(* CoDeSys 2.3.9.31 project: myhome.pro *)
(* Libraries: TcSUPS.lib 22.3.10 14:59:22, TcBaseMath.lib 27.7.04 13:07:56, TcMath.lib 23.9.04 16:15:30, TcBABasic.lib 29.5.12 16:01:34, TcBase.lib 14.5.09 13:14:08, TcSystem.lib 27.2.12 16:08:36, TcUtilities.lib 2.3.12 20:25:40, TcEL6851.lib 22.4.12 13:04:27, STANDARD.LIB 5.6.98 13:03:02, TcpIp.lib 13.10.11 11:31:34, beckhoff_network_121.lib 6.5.14 22:11:45, oscat_basic_333.lib 6.5.14 22:41:24 *)

(* Global variable list: Global_Variables *)
VAR_GLOBAL

	SYS_VKE_0:		BOOL	:=	FALSE;		(*SYSTEM ALWAYS 0*)
	SYS_VKE_1:		BOOL	:=	TRUE;		(*SYSTEM ALWAYS 1*)
	SYS_IBN_1:		BOOL	:=	TRUE;		(*SYSTEM IBN ALWAYS 1*)

	di_System_Time:	DINT;

	SYS_FPE_100MS:	BOOL	:=	FALSE;		(*SYSTEM TIME 0.1 sec*)
	SYS_FPE_200MS:	BOOL	:=	FALSE;		(*SYSTEM TIME 0.2 sec*)
	SYS_FPE_500MS:	BOOL	:=	FALSE;		(*SYSTEM TIME 0.5 sec*)
	SYS_FPE_1S:		BOOL	:=	FALSE;		(*SYSTEM TIME 1.0 sec*)
	SYS_FPE_2S:		BOOL	:=	FALSE;		(*SYSTEM TIME 2.0 sec*)

	SYS_TOG_100MS:	BOOL	:=	FALSE;		(*SYSTEM TIME 0.1 sec*)
	SYS_TOG_200MS:	BOOL	:=	FALSE;		(*SYSTEM TIME 0.2 sec*)
	SYS_TOG_500MS:	BOOL	:=	FALSE;		(*SYSTEM TIME 0.5 sec*)
	SYS_TOG_1S:		BOOL	:=	FALSE;		(*SYSTEM TIME 1.0 sec*)
	SYS_TOG_2S:		BOOL	:=	FALSE;		(*SYSTEM TIME 2.0 sec*)

	SYS_T_100MS:		TON;					(*SYSTEM TIME 0.1 sec*)
	SYS_T_200MS:		TON;					(*SYSTEM TIME 0.2 sec*)
	SYS_T_500MS:		TON;					(*SYSTEM TIME 0.5 sec*)
	SYS_T_1S:			TON;					(*SYSTEM TIME 1.0 sec*)
	SYS_T_2S:			TON;					(*SYSTEM TIME 2.0 sec*)

	AX_FPE_100MS:	R_TRIG;				(*SYSTEM AUX FPE 0.1 sec*)
	AX_FPE_200MS:	R_TRIG;				(*SYSTEM AUX FPE 0.2 sec*)
	AX_FPE_500MS:	R_TRIG;				(*SYSTEM AUX FPE 0.5 sec*)
	AX_FPE_1S:		R_TRIG;				(*SYSTEM AUX FPE 1.0 sec*)
	AX_FPE_2S:		R_TRIG;				(*SYSTEM AUX FPE 2.0 sec*)

(*DIGITAL INPUTS/Outputs*)
	(*SPS Switch 01 Arbeitsraum*)
	DI_S01_1 	AT %IX50.0 : BOOL;	(*Function Left 1*)
	DI_S01_2	AT %IX50.1 : BOOL;	(*Function Right 1*)
	DI_S01_3	AT %IX50.2 : BOOL;	(*Function Left 2*)
	DI_S01_4	AT %IX50.3 : BOOL;	(*Function Right 2*)
	DI_S01_5	AT %IX50.4 : BOOL;	(*Function Left 3*)
	DI_S01_6	AT %IX50.5 : BOOL;	(*Function Right 3*)
	DO_S01_0 	AT %QX50.0 : BOOL;	(*Status LED Left 1*)
	DO_S01_1 	AT %QX50.1 : BOOL;	(*Status LED Right 1*)
	DO_S01_2 	AT %QX50.2 : BOOL;	(*Status LED Left 2*)
	DO_S01_3 	AT %QX50.3 : BOOL;	(*Status LED Right 2*)
	DO_S01_4 	AT %QX50.4 : BOOL;	(*Status LED Left 3*)
	DO_S01_5 	AT %QX50.5 : BOOL;	(*Status LED Right 3*)
	DO_S01_6 	AT %QX50.6 : BOOL;	(*Background LED*)

	(*SPS Switch 02 Wohnzimmer*)
	DI_S02_1 	AT %IX50.6 : BOOL;	(*Function Left 1*)
	DI_S02_2	AT %IX50.7 : BOOL;	(*Function Right 1*)
	DI_S02_3	AT %IX51.0 : BOOL;	(*Function Left 2*)
	DI_S02_4	AT %IX51.1 : BOOL;	(*Function Right 2*)
	DI_S02_5	AT %IX51.2 : BOOL;	(*Function Left 3*)
	DI_S02_6	AT %IX51.3 : BOOL;	(*Function Right 3*)
	DO_S02_0 	AT %QX50.7 : BOOL;	(*Status LED Left 1*)
	DO_S02_1 	AT %QX51.0 : BOOL;	(*Status LED Right 1*)
	DO_S02_2 	AT %QX51.1 : BOOL;	(*Status LED Left 2*)
	DO_S02_3 	AT %QX51.2 : BOOL;	(*Status LED Right 2*)
	DO_S02_4 	AT %QX51.3 : BOOL;	(*Status LED Left 3*)
	DO_S02_5 	AT %QX51.4 : BOOL;	(*Status LED Right 3*)
	DO_S02_6 	AT %QX51.5 : BOOL;	(*Background LED*)

	(*DOUBLE Switch 03*)
	DI_S03_1 	AT %IX51.4 : BOOL;	(*Function Left*)
	DI_S03_2 	AT %IX51.5 : BOOL;	(*Function Right*)

	(*DOUBLE Switch 04*)
	DI_S04_1 	AT %IX51.6 : BOOL;	(*Function Left*)
	DI_S04_2 	AT %IX51.7 : BOOL;	(*Function Right*)

	(*SPS Switch 05 Schlafzimmer Bett Links*)
	DI_S05_1 	AT %IX52.0 : BOOL;	(*Function Left 1*)
	DI_S05_2	AT %IX52.1 : BOOL;	(*Function Right 1*)
	DI_S05_3	AT %IX52.2 : BOOL;	(*Function Left 2*)
	DI_S05_4	AT %IX52.3 : BOOL;	(*Function Right 2*)
	DI_S05_5	AT %IX52.4 : BOOL;	(*Function Left 3*)
	DI_S05_6	AT %IX52.5 : BOOL;	(*Function Right 3*)
	DO_S05_0 	AT %QX51.6 : BOOL;	(*Status LED Left 1*)
	DO_S05_1 	AT %QX51.7 : BOOL;	(*Status LED Right 1*)
	DO_S05_2 	AT %QX52.0 : BOOL;	(*Status LED Left 2*)
	DO_S05_3 	AT %QX52.1 : BOOL;	(*Status LED Right 2*)
	DO_S05_4 	AT %QX52.2 : BOOL;	(*Status LED Left 3*)
	DO_S05_5 	AT %QX52.3 : BOOL;	(*Status LED Right 3*)
	DO_S05_6 	AT %QX52.4 : BOOL;	(*Background LED*)

	(*SPS Switch 06 Schlafzimmer Bett Rechts*)
	DI_S06_1 	AT %IX52.6 : BOOL;	(*Function Left 1*)
	DI_S06_2	AT %IX52.7 : BOOL;	(*Function Right 1*)
	DI_S06_3	AT %IX53.0 : BOOL;	(*Function Left 2*)
	DI_S06_4	AT %IX53.1 : BOOL;	(*Function Right 2*)
	DI_S06_5	AT %IX53.2 : BOOL;	(*Function Left 3*)
	DI_S06_6	AT %IX53.3 : BOOL;	(*Function Right 3*)
	DO_S06_0 	AT %QX52.5 : BOOL;	(*Status LED Left 1*)
	DO_S06_1 	AT %QX52.6 : BOOL;	(*Status LED Right 1*)
	DO_S06_2 	AT %QX52.7 : BOOL;	(*Status LED Left 2*)
	DO_S06_3 	AT %QX53.0 : BOOL;	(*Status LED Right 2*)
	DO_S06_4 	AT %QX53.1 : BOOL;	(*Status LED Left 3*)
	DO_S06_5 	AT %QX53.2 : BOOL;	(*Status LED Right 3*)
	DO_S06_6 	AT %QX53.3 : BOOL;	(*Background LED*)

	(*DOUBLE Switch 07*)
	DI_S07_1 	AT %IX53.4 : BOOL;	(*Function Left*)
	DI_S07_2 	AT %IX53.5 : BOOL;	(*Function Right*)

	(*SINGLE Switch 08*)
	DI_S08	 	AT %IX53.6 : BOOL;	(*Function*)

	(*SINGLE Switch 09*)
	DI_S09	 	AT %IX53.7 : BOOL;	(*Function*)

	(*SINGLE Switch 10*)
	DI_S10	 	AT %IX54.0 : BOOL;	(*Function*)

	(*SINGLE Swith 11*)
	DI_S11	 	AT %IX54.1 : BOOL;	(*Function*)

	(*Relais*)
	DO_NN_K01	AT %QX54.0 : BOOL;	(*Relais Netzteil Arbeitsraum*)
	DO_NN_K02	AT %QX54.1 : BOOL;	(*Relais Steckdosen Arbeitsraum*)
	DO_NN_K03	AT %QX54.2 : BOOL;	(*Relais Netzteil Wohnzimmer*)
	DO_NN_K04	AT %QX54.3 : BOOL;	(*Relais Steckdosen Fernseher*)
	DO_NN_K05	AT %QX54.4 : BOOL;	(*Relais Netzteil Küche*)
	DO_NN_K06	AT %QX54.5 : BOOL;	(*Relais Netzteil Zimmer / Schlafzimmer*)
	DO_NN_K07	AT %QX54.6 : BOOL;	(*Relais Netzteil WC, Gang und Abstellraum*)
	DO_NN_K08	AT %QX54.7 : BOOL;	(*Relais Reserve*)
	DO_NN_K09	AT %QX53.6 : BOOL;	(*Relais Reserve*)
	DO_NN_K10	AT %QX53.7 : BOOL;	(*Relais Reserve*)

(* DMX Line *)
	fbEL6851Communication	:	FB_EL6851Communication;
	stDMXInDataLinie01               AT %I*	:	ST_EL6851InData;
	stDMXOutDataLinie01              AT %Q*	:	ST_EL6851OutData;
	stCommandBuffer01						:	ST_DMXCommandBuffer;
	arrDMXProcessData						:	ARRAY [1..512] OF BYTE;

END_VAR

(* Global variable list: TwinCAT_Configuration *)
(* Generated automatically by TwinCAT - (read only) *)
VAR_CONFIG
	.stDMXInDataLinie01 AT %IB56 : ST_EL6851InData;
	.stDMXOutDataLinie01 AT %QB56 : ST_EL6851OutData;
END_VAR

(* Data type *)
TYPE Type_HSV :
STRUCT
	Hue	:			REAL;
	Saturation:		REAL:= 100.0;
	Brightness:		REAL:=100.0;
END_STRUCT
END_TYPE

(* Data type *)
TYPE Type_LED :
STRUCT
	Switch_ON:			BOOL;
	Switch_RANDOM:		BOOL;
	bLight:				BOOL;
	Config:				Type_LED_CONFIG;
	Value:				REAL:=100;
	Brightness:			BYTE;
	fbDimmer2Switch: FB_Dimmer2Switch;
	fpSwitchOnOff: F_TRIG;
END_STRUCT
END_TYPE

(* Data type *)
TYPE Type_LED_CONFIG :
STRUCT
	tDimmTime: 		REAL	:= 5000;
	bDimmOnMode:	BOOL	:= TRUE;
	tDimmOnTime:		REAL	:= 500;
	bDimmOffMode:	BOOL	:= TRUE;
	tDimmOffTime:		REAL	:= 1000;
	Brightness_MAX	:REAL:=255;
END_STRUCT
END_TYPE

(* Data type *)
TYPE Type_LED_RGB :
STRUCT
	Hue				:REAL;
	Saturation			:REAL:= 100.0;
	Brightness			:REAL:=100;
	Switch_ON			:BOOL;
	Switch_RANDOM	:BOOL;
	bLight:			BOOL;
	Config				:Type_LED_RGB_CONFIG;
	Red					:BYTE;
	Green				:BYTE;
	Blue					:BYTE;
	fbDimmer2Switch: FB_Dimmer2Switch;
	fpSwitchOnOff: F_TRIG;
END_STRUCT
END_TYPE

(* Data type *)
TYPE Type_LED_RGB_CONFIG :
STRUCT
	Speed_RANDOM	:REAL;

	tDimmTime: 		REAL	:= 5000;
	bDimmOnMode:	BOOL	:= TRUE;
	tDimmOnTime:		REAL	:= 500;
	bDimmOffMode:	BOOL	:= TRUE;
	tDimmOffTime:		REAL	:= 1000;
END_STRUCT
END_TYPE

(* Data type *)
TYPE Type_SCENE_CONFIG :
STRUCT
	tDimmTime: 		REAL	:= 5000;
	bDimmOnMode:	BOOL	:= TRUE;
	tDimmOnTime:		REAL	:= 500;
	bDimmOffMode:	BOOL	:= TRUE;
	tDimmOffTime:		REAL	:= 1000;
END_STRUCT
END_TYPE

(* Data type *)
TYPE Type_SCENE_WZ :
STRUCT
	bSceneActive:			BOOL;
	byWhiteUpNorth:			BYTE;
	byWhiteUpWest:			BYTE;
	byWhiteUpSouthEast:		BYTE;
	byWhiteMiddleNorthWest:	BYTE;
	byWhiteMiddleSouthEast:	BYTE;
	byWhiteDownNorthWest:	BYTE;
	byWhiteDownSouthEast:	BYTE;
	tyHSVUp:				Type_HSV;
	tyHSVMiddle: 			Type_HSV;
	tyHSVDown: 				Type_HSV;
	tyConfig:					Type_SCENE_CONFIG;
END_STRUCT
END_TYPE

(* POU MAIN, ST *)
PROGRAM MAIN
VAR
	YahooWeatherAltlengbach: FB_WEATHER;
END_VAR
FC_00_BASICS();

(*Aufruf Wohnräume*)
FC_01_ARBEITSZIMMER();
FC_02_WOHNZIMMER();
FC_03_KUECHE();
FC_04_ZIMMER();
FC_05_WC_GANG();

(*YahooWeatherAltlengbach();*)

(*WORLD_WEATHER_test();*)
YAHOO_WEATHER_test();

fbEL6851Communication(	wSourceManufacturerID := 16#42_41,
						dwSourceDeviceID := 16#12_13_14_15,
						bEnableSendingData := TRUE,
						bSetCycleMode := TRUE,
						bSendDefaultData := FALSE,
						uiDataLength := 512,
						dwOptions := 0,
						stEL6851InData := stDMXInDataLinie01,
						stEL6851OutData := stDMXOutDataLinie01,
						stCommandBuffer := stCommandBuffer01,
						arrProcessData := arrDMXProcessData);
END_PROGRAM

(* POU Weather/FB_WEATHER, ST *)
FUNCTION_BLOCK FB_WEATHER
VAR_INPUT
END_VAR
VAR_OUTPUT
END_VAR
VAR
	FB_Weather_PLZ_3033: YAHOO_WEATHER;
	vBOOL: BOOL := FALSE;
	vIP_C : IP_C;
	vS_BUF : NETWORK_BUFFER;
	vR_BUF : NETWORK_BUFFER;
	vYW : YAHOO_WEATHER_DATA;
	vBUSY : BOOL;
	vDONE : BOOL;
	vERROR_C : DWORD;
	vERROR_T : BYTE;
END_VAR
FB_Weather_PLZ_3033(
	ACTIVATE:= vBOOL,
	UNITS:= FALSE,
	LOCATION:= '541490',
	IP_C:=vIP_C ,
	S_BUF:=vS_BUF ,
	R_BUF:=vR_BUF ,
	YW:= vYW,
	BUSY=> vBUSY,
	DONE=>vDONE ,
	ERROR_C=>vERROR_C ,
	ERROR_T=>vERROR_T );
END_FUNCTION_BLOCK

(* POU FC_00_BASICS, ST *)
PROGRAM FC_00_BASICS
VAR
	T_100ms_TON: TON;
	T_100ms_TOF: TOF;

(* UPS related ... *)
	fbUPS			: FB_S_UPS;			(* UPS-FB instance *)
					(* Default Values of FB_S_UPS-Inputs:
						sNetID 			:= '' ==> local netid
						iPLCPort 		:= AMSPORT_R0_PLC_RTS1 ==> 801 = 1st Runtime System
						iUPSPort		:= 16#4A8 ==> Port for reading Power State of UPS
						tTimeout 		:= DEFAULT_ADS_TIMEOUT ==> 5S
						eUpsMode 		:= eSUPS_WrPersistData_Shutdown ==> writing persistent data + shutdown
						ePersistentMode := SPDM_2PASS ==> All data is from same plc cycle, cycletime exceeds possible. Plc stops with the shutdown, a few cycles after writing persistent data. 
						tRecoverTime 	:= T#10s ==> 10s power to recover from short power failure before eSUPS_PowerOK is reported (in mode eSUPS_WrPersistData_NoShutdown/eSUPS_CheckPowerStatus)
					*)
	eUpsMode		: E_S_UPS_Mode	:= eSUPS_WrPersistData_Shutdown; (* UPS mode (writing persistent data + shutdown) *)

	(* !!! TO DO: REPLACE WITH YOUR PLC VARIABLES/FB INSTANCES !!! regular PLC variables/FB instances ... *)
	iCounter		: UDINT;					(* non persistent counter *)

END_VAR

VAR PERSISTENT
	(* !!! TO DO: REPLACE WITH YOUR PERSISTENT PLC VARIABLES !!! persistent variables ... *)
	iPowerFailureCount: UDINT:=0; (* persistent counter of power failures *)
END_VAR
SYS_VKE_0		:=	FALSE;
SYS_VKE_1		:=	TRUE;
SYS_IBN_1		:=	TRUE;

di_System_Time := TIME_TO_DINT(TIME());


(*GENERATE SYSTEM PULSE FLAGS*)

SYS_T_100MS(IN:= SYS_IBN_1 AND NOT SYS_T_100MS.Q, PT:= T#100MS);
SYS_T_200MS(IN:= SYS_IBN_1 AND NOT SYS_T_200MS.Q, PT:= T#200MS);
SYS_T_500MS(IN:= SYS_IBN_1 AND NOT SYS_T_500MS.Q, PT:= T#500MS);
SYS_T_1S(IN:= SYS_IBN_1 AND NOT SYS_T_1S.Q, PT:= T#1S);
SYS_T_2S(IN:= SYS_IBN_1 AND NOT SYS_T_2S.Q, PT:= T#2S);

IF SYS_T_100MS.Q	THEN
	IF SYS_TOG_100MS THEN
		SYS_TOG_100MS := FALSE; 	ELSE	SYS_TOG_100MS := TRUE;
	END_IF
END_IF

IF SYS_T_200MS.Q	THEN
	IF SYS_TOG_200MS THEN
		SYS_TOG_200MS := FALSE; 	ELSE	SYS_TOG_200MS := TRUE;
	END_IF
END_IF

IF SYS_T_500MS.Q	THEN
	IF SYS_TOG_500MS THEN
		SYS_TOG_500MS := FALSE; 	ELSE	SYS_TOG_500MS := TRUE;
	END_IF
END_IF

IF SYS_T_1S.Q	THEN
	IF SYS_TOG_1S THEN
		SYS_TOG_1S := FALSE; 	ELSE	SYS_TOG_1S := TRUE;
	END_IF
END_IF

IF SYS_T_2S.Q	THEN
	IF SYS_TOG_2S THEN
		SYS_TOG_2S := FALSE; 	ELSE	SYS_TOG_2S := TRUE;
	END_IF
END_IF

AX_FPE_100MS(CLK:= SYS_TOG_100MS , Q=> SYS_FPE_100MS);
AX_FPE_200MS(CLK:= SYS_TOG_200MS , Q=> SYS_FPE_200MS);
AX_FPE_500MS(CLK:= SYS_TOG_500MS , Q=> SYS_FPE_500MS);
AX_FPE_1S(CLK:= SYS_TOG_1S , Q=> SYS_FPE_1S);
AX_FPE_2S(CLK:= SYS_TOG_2S , Q=> SYS_FPE_2S);

(* S-UPS Demo *)

(* call UPS-FB instance in first lines of the fastest PLC Task *)
fbUPS(eUpsMode := eUpsMode);
(* eUpsMode =							in case of powerfailure:
	 eSUPS_WrPersistData_Shutdown 		 	writing of persistent data + shutdown
	 eSUPS_WrPersistData_NoShutdown 		writing of PERSISTENT data, no shutdown
	 eSUPS_CheckPowerStatus 				reports powerfailure without ACTION (no writing, no shutdown) 
	 eSUPS_ImmediateShutdown 				skips writing of data, immediate shutdown
*)

(* evaluate UPS State *)
IF eGlobalSUpsState = eSUPS_PowerFailure THEN
	(* first cycle of powerfailure *)

	(* execute code that should only be done once with each powerfailure, i.e. increase powerfailure counter *)
	iPowerFailureCount := iPowerFailureCount + 1;
END_IF
END_PROGRAM

(* POU FC_01_ARBEITSZIMMER, ST *)
PROGRAM FC_01_ARBEITSZIMMER
VAR PERSISTENT
	tyWhiteCeiling:			Type_LED;
	tyWhiteWorkplace:		Type_LED;
	tyWhiteRegal:			Type_LED;
	tyWhiteAbstellraum:		Type_LED;
	tyWhiteReserve1:			Type_LED;
	tyWhiteReserve2:			Type_LED;
	tyWhiteReserve3:			Type_LED;
	tyWhiteReserve4:			Type_LED;
END_VAR
(*LED light white ceiling*)
PRG_LED_SINGLECOLOR(
	i_bSwitchOn:= DI_S01_1,
	i_bSwitchOff:= FALSE,
	i_bSwitchOnOff:= DI_S01_1,
	i_iSceneValue:= ,
	io_TypeLED:= tyWhiteCeiling);

(*LED light white workplace*)
PRG_LED_SINGLECOLOR(
	i_bSwitchOn:= DI_S01_1,
	i_bSwitchOff:= FALSE,
	i_bSwitchOnOff:= FALSE,
	i_iSceneValue:= ,
	io_TypeLED:= tyWhiteWorkplace);

(*LED light white Regal*)
PRG_LED_SINGLECOLOR(
	i_bSwitchOn:= FALSE,
	i_bSwitchOff:= FALSE,
	i_bSwitchOnOff:= FALSE,
	i_iSceneValue:= ,
	io_TypeLED:= tyWhiteRegal);

(*LED light white Abstellraum*)
PRG_LED_SINGLECOLOR(
	i_bSwitchOn:= FALSE,
	i_bSwitchOff:= FALSE,
	i_bSwitchOnOff:= FALSE,
	i_iSceneValue:= ,
	io_TypeLED:= tyWhiteAbstellraum);

(*LED light white Reserve*)
PRG_LED_SINGLECOLOR(
	i_bSwitchOn:= FALSE,
	i_bSwitchOff:= FALSE,
	i_bSwitchOnOff:= FALSE,
	i_iSceneValue:= ,
	io_TypeLED:= tyWhiteReserve1);

(*LED light white Reserve*)
PRG_LED_SINGLECOLOR(
	i_bSwitchOn:= FALSE,
	i_bSwitchOff:= FALSE,
	i_bSwitchOnOff:= FALSE,
	i_iSceneValue:= ,
	io_TypeLED:= tyWhiteReserve2);

(*LED light white Reserve*)
PRG_LED_SINGLECOLOR(
	i_bSwitchOn:= FALSE,
	i_bSwitchOff:= FALSE,
	i_bSwitchOnOff:= FALSE,
	i_iSceneValue:= ,
	io_TypeLED:= tyWhiteReserve3);

(*LED light white Reserve*)
PRG_LED_SINGLECOLOR(
	i_bSwitchOn:= FALSE,
	i_bSwitchOff:= FALSE,
	i_bSwitchOnOff:= FALSE,
	i_iSceneValue:= ,
	io_TypeLED:= tyWhiteReserve4);

(*relay for power supply*)
DO_NN_K01 :=	tyWhiteCeiling.bLight OR tyWhiteWorkplace.bLight OR tyWhiteRegal.bLight OR
				tyWhiteAbstellraum.bLight OR tyWhiteReserve1.bLight OR tyWhiteReserve2.bLight OR
				tyWhiteReserve3.bLight OR tyWhiteReserve4.bLight;
(*DMX communication*)
arrDMXProcessData[1] := tyWhiteCeiling.Brightness;
arrDMXProcessData[2] := tyWhiteWorkplace.Brightness;
arrDMXProcessData[3] := tyWhiteRegal.Brightness;
arrDMXProcessData[4] := tyWhiteAbstellraum.Brightness;
arrDMXProcessData[5] := tyWhiteReserve1.Brightness;
arrDMXProcessData[6] := tyWhiteReserve2.Brightness;
arrDMXProcessData[7] := tyWhiteReserve3.Brightness;
arrDMXProcessData[8] := tyWhiteReserve4.Brightness;
END_PROGRAM

(* POU PRG_LED_SINGLECOLOR, ST *)
PROGRAM PRG_LED_SINGLECOLOR
VAR_INPUT
	i_bSwitchOn:		BOOL;
	i_bSwitchOff:		BOOL;
	i_bSwitchOnOff:	BOOL;
	i_iSceneValue:	INT;
END_VAR

VAR_IN_OUT
	io_TypeLED: Type_LED;		(*CONTAINS THE LIGHT STATUS*)
END_VAR
(*flag positive edge of switch for on and off*)
io_TypeLED.fpSwitchOnOff(CLK:= i_bSwitchOnOff );

(*switch light on*)
IF i_bSwitchOn OR (io_TypeLED.fpSwitchOnOff.Q AND NOT io_TypeLED.bLight) THEN
	io_TypeLED.Switch_ON := TRUE;
END_IF

(*switch light off*)
IF i_bSwitchOff OR (io_TypeLED.fpSwitchOnOff.Q AND io_TypeLED.bLight) THEN
	io_TypeLED.Switch_ON := FALSE;
END_IF

io_TypeLED.fbDimmer2Switch(
	bSwitchDimmUp:= FALSE,
	bSwitchDimmDown:= FALSE,
	bOn:= io_TypeLED.Switch_ON,
	bOff:= NOT io_TypeLED.Switch_ON,
	bSetDimmValue:= FALSE,
	nDimmValue:= 0,
	tSwitchOverTime:=T#300MS ,
	tDimmTime:= REAL_TO_TIME(io_TypeLED.Config.tDimmTime),
	bMemoryModeOn:= TRUE,
	nOnValueWithoutMemoryMode:= 0,
	bDimmOnMode:= io_TypeLED.Config.bDimmOnMode,
	tDimmOnTime:= REAL_TO_TIME(io_TypeLED.Config.tDimmOnTime),
	bDimmOffMode:= io_TypeLED.Config.bDimmOffMode,
	tDimmOffTime:= REAL_TO_TIME(io_TypeLED.Config.tDimmOffTime),
	nOutMin:= 0,
	nOutMax:=100,
	bLight=> io_TypeLED.bLight);

io_TypeLED.Brightness := REAL_TO_BYTE(UINT_TO_REAL(io_TypeLED.fbDimmer2Switch.nOut)/100*io_TypeLED.Config.Brightness_MAX*(io_TypeLED.Value/100));
END_PROGRAM

(* POU FC_02_WOHNZIMMER, ST *)
PROGRAM FC_02_WOHNZIMMER
VAR PERSISTENT
	tyScene1: Type_SCENE_WZ;
	tyScene2: Type_SCENE_WZ;
	tyScene3: Type_SCENE_WZ;
	tyScene4: Type_SCENE_WZ;
	tyScene5: Type_SCENE_WZ;
	tyScene6: Type_SCENE_WZ;
	tyScene7: Type_SCENE_WZ;
	tyScene8: Type_SCENE_WZ;
	tyScene9: Type_SCENE_WZ;
	tyScene10: Type_SCENE_WZ;
	tyScene11: Type_SCENE_WZ;
	tyScene12: Type_SCENE_WZ;
	tyScene13: Type_SCENE_WZ;
	tyScene14: Type_SCENE_WZ;
	tyScene15: Type_SCENE_WZ;

	tyActScene:Type_SCENE_WZ;

	tyWhiteUpNorth:				Type_LED;
	tyWhiteUpWest:				Type_LED;
	tyWhiteUpSouthEast:			Type_LED;
	tyWhiteMiddleNorthWest:		Type_LED;
	tyWhiteMiddleSouthEast:		Type_LED;
	tyWhiteDownNorthWest:		Type_LED;
	tyWhiteDownSouthEast:		Type_LED;
	tyRGBUp:					Type_LED_RGB;
	tyRGBMiddle: 				Type_LED_RGB;
	tyRGBDown: 					Type_LED_RGB;

END_VAR
(*Scene control*)
PRG_SCENE_CONTROL_WZ(
	i_bNextScene:= , 
	i_bPrevScene:= , 
	io_tyScene1:= tyScene1,
	io_tyScene2:= tyScene2,
	io_tyScene3:= tyScene3,
	io_tyScene4:= tyScene4,
	io_tyScene5:= tyScene5,
	io_tyScene6:= tyScene6,
	io_tyScene7:= tyScene7,
	io_tyScene8:= tyScene8,
	io_tyScene9:= tyScene9,
	io_tyScene10:= tyScene10,
	io_tyScene11:= tyScene11,
	io_tyScene12:= tyScene12,
	io_tyScene13:= tyScene13,
	io_tyScene14:= tyScene14,
	io_tyScene15:= tyScene15,
	o_tyActScene=> tyActScene);

(*LED light white up north*)
PRG_LED_SINGLECOLOR(
	i_bSwitchOn:= FALSE,
	i_bSwitchOff:= FALSE,
	i_bSwitchOnOff:= FALSE,
	i_iSceneValue:= tyActScene.byWhiteUpNorth,
	io_TypeLED:= tyWhiteUpNorth);

(*LED light white up west*)
PRG_LED_SINGLECOLOR(
	i_bSwitchOn:= FALSE,
	i_bSwitchOff:= FALSE,
	i_bSwitchOnOff:= FALSE,
	i_iSceneValue:= tyActScene.byWhiteUpWest,
	io_TypeLED:= tyWhiteUpWest);

(*LED light white up southeast*)
PRG_LED_SINGLECOLOR(
	i_bSwitchOn:= FALSE,
	i_bSwitchOff:= FALSE,
	i_bSwitchOnOff:=FALSE ,
	i_iSceneValue:= tyActScene.byWhiteUpSouthEast,
	io_TypeLED:= tyWhiteUpSouthEast);

(*LED light white middle northwest*)
PRG_LED_SINGLECOLOR(
	i_bSwitchOn:= FALSE,
	i_bSwitchOff:= FALSE,
	i_bSwitchOnOff:= FALSE,
	i_iSceneValue:= tyActScene.byWhiteMiddleNorthWest,
	io_TypeLED:= tyWhiteMiddleNorthWest);

(*LED light white middle southeast*)
PRG_LED_SINGLECOLOR(
	i_bSwitchOn:= FALSE,
	i_bSwitchOff:= FALSE,
	i_bSwitchOnOff:= FALSE,
	i_iSceneValue:= tyActScene.byWhiteMiddleSouthEast,
	io_TypeLED:= tyWhiteMiddleSouthEast);

(*LED light white down northwest*)
PRG_LED_SINGLECOLOR(
	i_bSwitchOn:= FALSE,
	i_bSwitchOff:= FALSE,
	i_bSwitchOnOff:=FALSE ,
	i_iSceneValue:= tyActScene.byWhiteDownNorthWest,
	io_TypeLED:= tyWhiteDownNorthWest);

(*LED light white down southeast*)
PRG_LED_SINGLECOLOR(
	i_bSwitchOn:= FALSE,
	i_bSwitchOff:= FALSE,
	i_bSwitchOnOff:= FALSE,
	i_iSceneValue:= tyActScene.byWhiteDownSouthEast,
	io_TypeLED:= tyWhiteDownSouthEast);

(*LED light RGB upper row*)
PRG_LED_MULTICOLOR(
	i_SwitchON:= FALSE,
	i_SwitchOFF:= FALSE,
	i_bSwitchOnOff:= DI_S02_3,
	i_iSceneValue:= ,
	di_SysTime:= di_System_Time,
	io_Type_LED_RGB:= tyRGBUp);

(*LED light RGB middle row*)
PRG_LED_MULTICOLOR(
	i_SwitchON:= FALSE,
	i_SwitchOFF:= FALSE,
	i_bSwitchOnOff:= FALSE,
	i_iSceneValue:= ,
	di_SysTime:= di_System_Time,
	io_Type_LED_RGB:= tyRGBMiddle);

(*LED light RGB bottom row*)
PRG_LED_MULTICOLOR(
	i_SwitchON:= FALSE,
	i_SwitchOFF:= FALSE,
	i_bSwitchOnOff:= FALSE,
	i_iSceneValue:= ,
	di_SysTime:=di_System_Time ,
	io_Type_LED_RGB:= tyRGBDown);

(*relay for power supply*)
DO_NN_K03:=	tyWhiteUpNorth.bLight OR tyWhiteUpWest.bLight OR tyWhiteUpSouthEast.bLight OR
				tyWhiteMiddleNorthWest.bLight OR tyWhiteMiddleSouthEast.bLight OR tyWhiteDownNorthWest.bLight OR
				tyWhiteDownSouthEast.bLight OR tyRGBUp.bLight OR tyRGBMiddle.bLight OR tyRGBDown.bLight;

(*DMX communication*)
arrDMXProcessData[10] := tyWhiteUpNorth.Brightness;
arrDMXProcessData[11] := tyWhiteUpWest.Brightness;
arrDMXProcessData[12] := tyWhiteUpSouthEast.Brightness;
arrDMXProcessData[13] := tyWhiteMiddleNorthWest.Brightness;
arrDMXProcessData[14] := tyWhiteMiddleSouthEast.Brightness;
arrDMXProcessData[15] := tyWhiteDownNorthWest.Brightness;
arrDMXProcessData[16] := tyWhiteDownSouthEast.Brightness;
arrDMXProcessData[17] := tyRGBUp.Red;
arrDMXProcessData[18] := tyRGBUp.Green;
arrDMXProcessData[19] := tyRGBUp.Blue;
arrDMXProcessData[20] := tyRGBMiddle.Red;
arrDMXProcessData[21] := tyRGBMiddle.Green;
arrDMXProcessData[22] := tyRGBMiddle.Blue;
arrDMXProcessData[23] := tyRGBDown.Red;
arrDMXProcessData[24] := tyRGBDown.Green;
arrDMXProcessData[25] := tyRGBDown.Blue;
END_PROGRAM

(* POU PRG_SCENE_CONTROL_WZ, ST *)
PROGRAM PRG_SCENE_CONTROL_WZ
VAR_INPUT
	i_bNextScene:	BOOL;
	i_bPrevScene:	BOOL;
END_VAR

VAR_IN_OUT
	io_tyScene1: Type_SCENE_WZ;
	io_tyScene2: Type_SCENE_WZ;
	io_tyScene3: Type_SCENE_WZ;
	io_tyScene4: Type_SCENE_WZ;
	io_tyScene5: Type_SCENE_WZ;
	io_tyScene6: Type_SCENE_WZ;
	io_tyScene7: Type_SCENE_WZ;
	io_tyScene8: Type_SCENE_WZ;
	io_tyScene9: Type_SCENE_WZ;
	io_tyScene10: Type_SCENE_WZ;
	io_tyScene11: Type_SCENE_WZ;
	io_tyScene12: Type_SCENE_WZ;
	io_tyScene13: Type_SCENE_WZ;
	io_tyScene14: Type_SCENE_WZ;
	io_tyScene15: Type_SCENE_WZ;
END_VAR

VAR_OUTPUT
	o_tyActScene: Type_SCENE_WZ;
END_VAR

VAR
	fpNextScene: F_TRIG;
	fpPrevScene: F_TRIG;
	v_iActScene:	INT	:= 1;
END_VAR
fpNextScene(CLK:=i_bNextScene);
fpPrevScene(CLK:=i_bPrevScene);

IF fpNextScene.Q THEN
	v_iActScene := v_iActScene + 1;
END_IF

IF fpPrevScene.Q THEN
	v_iActScene := v_iActScene - 1;
END_IF

IF v_iActScene >= 17 THEN
	v_iActScene := 1;
END_IF

IF v_iActScene <= 0 THEN
	v_iActScene := 16;
END_IF

o_tyActScene := io_tyScene1;

CASE v_iActScene OF
1:	o_tyActScene := io_tyScene1;
2:	o_tyActScene := io_tyScene2;
3:	o_tyActScene := io_tyScene3;
4:	o_tyActScene := io_tyScene4;
5:	o_tyActScene := io_tyScene5;
6:	o_tyActScene := io_tyScene6;
7:	o_tyActScene := io_tyScene7;
8:	o_tyActScene := io_tyScene8;
9:	o_tyActScene := io_tyScene9;
10:	o_tyActScene := io_tyScene10;
11:	o_tyActScene := io_tyScene11;
12:	o_tyActScene := io_tyScene12;
13:	o_tyActScene := io_tyScene13;
14:	o_tyActScene := io_tyScene14;
15:	o_tyActScene := io_tyScene15;
END_CASE
END_PROGRAM

(* POU PRG_LED_MULTICOLOR, ST *)
PROGRAM PRG_LED_MULTICOLOR
VAR_INPUT
	i_SwitchON:	BOOL;
	i_SwitchOFF:	BOOL;
	i_bSwitchOnOff:	BOOL;
	i_iSceneValue:	INT;
	di_SysTime:	DINT;
END_VAR

VAR
	v_HUE: REAL;
	v_SATURATION: REAL;
	v_VALUE: REAL;
	v_RED: BYTE;
	v_GREEN: BYTE;
	v_BLUE: BYTE;
	v_VAR_H: REAL;
	v_VAR_I: REAL;
	v_VAR_1: REAL;
	v_VAR_2: REAL;
	v_VAR_3: REAL;
	v_VAR_R: REAL;
	v_VAR_G: REAL;
	v_VAR_B: REAL;
	v_Sys_Time_last_Call:	DINT;
	v_Cycle_Time:	DINT;

END_VAR
VAR_IN_OUT
	io_Type_LED_RGB: Type_LED_RGB;		(*CONTAINS THE LIGHT STATUS*)
END_VAR
(*Calculate the System Time between the last and the actual cycle for automatic color switching*)
v_Cycle_Time := di_SysTime - v_Sys_Time_last_Call;
v_Sys_Time_last_Call := di_SysTime;

(*flag positive edge of switch for on and off*)
io_Type_LED_RGB.fpSwitchOnOff(CLK:= i_bSwitchOnOff );

(*switch light on*)
IF i_SwitchON OR (io_Type_LED_RGB.fpSwitchOnOff.Q AND NOT io_Type_LED_RGB.bLight) THEN
	io_Type_LED_RGB.Switch_ON := TRUE;
END_IF

(*switch light off*)
IF i_SwitchOFF OR (io_Type_LED_RGB.fpSwitchOnOff.Q AND io_Type_LED_RGB.bLight) THEN
	io_Type_LED_RGB.Switch_ON := FALSE;
END_IF

(*control light with standard FB from Beckhoff BaBasic Library*)
io_Type_LED_RGB.fbDimmer2Switch(
	bSwitchDimmUp:= FALSE,
	bSwitchDimmDown:= FALSE,
	bOn:= io_Type_LED_RGB.Switch_ON,
	bOff:= NOT io_Type_LED_RGB.Switch_ON,
	bSetDimmValue:= FALSE,
	nDimmValue:= 0,
	tSwitchOverTime:=T#300MS ,
	tDimmTime:= REAL_TO_TIME(io_Type_LED_RGB.Config.tDimmTime),
	bMemoryModeOn:= TRUE,
	nOnValueWithoutMemoryMode:= 0,
	bDimmOnMode:= io_Type_LED_RGB.Config.bDimmOnMode,
	tDimmOnTime:= REAL_TO_TIME(io_Type_LED_RGB.Config.tDimmOnTime),
	bDimmOffMode:= io_Type_LED_RGB.Config.bDimmOffMode,
	tDimmOffTime:= REAL_TO_TIME(io_Type_LED_RGB.Config.tDimmOffTime),
	nOutMin:= 0,
	nOutMax:=REAL_TO_UINT( io_Type_LED_RGB.Brightness),
	bLight=> io_Type_LED_RGB.bLight);

IF io_Type_LED_RGB.Config.Speed_RANDOM < 1000 THEN
	io_Type_LED_RGB.Config.Speed_RANDOM := 1000;
END_IF

IF io_Type_LED_RGB.Switch_RANDOM THEN
	io_Type_LED_RGB.Hue := io_Type_LED_RGB.Hue + 360/(io_Type_LED_RGB.Config.Speed_RANDOM)*DINT_TO_REAL(v_Cycle_Time);

	IF io_Type_LED_RGB.Hue >= 360 THEN
		io_Type_LED_RGB.Hue := io_Type_LED_RGB.Hue-360;
	END_IF
	IF io_Type_LED_RGB.Hue < 0 THEN
		io_Type_LED_RGB.Hue := 0;
	END_IF
END_IF

v_HUE := io_Type_LED_RGB.Hue / 360;
v_SATURATION := io_Type_LED_RGB.Saturation / 100;
v_VALUE := (io_Type_LED_RGB.Brightness*UINT_TO_REAL(io_Type_LED_RGB.fbDimmer2Switch.nOut)/100) / 100;

IF v_SATURATION = 0 THEN
	v_RED := REAL_TO_BYTE(v_VALUE * 255);
	v_GREEN := REAL_TO_BYTE(v_VALUE * 255);
	v_BLUE := REAL_TO_BYTE(v_VALUE * 255);
ELSE
	v_VAR_H := v_HUE * 6;
	v_VAR_I := FLOOR(REAL_TO_LREAL(v_VAR_H));
	v_VAR_1:= v_VALUE * (1 - v_SATURATION);
	v_VAR_2:= v_VALUE * (1 - v_SATURATION * (v_VAR_H - v_VAR_I));
	v_VAR_3:= v_VALUE * (1 - v_SATURATION * (1 - (v_VAR_H - v_VAR_I)));

	CASE REAL_TO_INT(v_VAR_I) OF
	0:
		v_VAR_R := v_VALUE;
		v_VAR_G := v_VAR_3;
		v_VAR_B := v_VAR_1;
	1:
		v_VAR_R := v_VAR_2;
		v_VAR_G := v_VALUE;
		v_VAR_B := v_VAR_1;
	2:
		v_VAR_R := v_VAR_1;
		v_VAR_G := v_VALUE;
		v_VAR_B := v_VAR_3;
	3:
		v_VAR_R := v_VAR_1;
		v_VAR_G := v_VAR_2;
		v_VAR_B := v_VALUE;
	4:
		v_VAR_R := v_VAR_3;
		v_VAR_G := v_VAR_1;
		v_VAR_B := v_VALUE;
	ELSE
		v_VAR_R := v_VALUE;
		v_VAR_G := v_VAR_1;
		v_VAR_B := v_VAR_2;
	END_CASE

	v_RED := REAL_TO_BYTE(v_VAR_R * 255);
	v_GREEN := REAL_TO_BYTE(v_VAR_G * 255);
	v_BLUE := REAL_TO_BYTE(v_VAR_B * 255);
END_IF

io_Type_LED_RGB.Red := v_RED;
io_Type_LED_RGB.Green := v_GREEN;
io_Type_LED_RGB.Blue := v_BLUE;
END_PROGRAM

(* POU FC_03_KUECHE, ST *)
PROGRAM FC_03_KUECHE
VAR PERSISTENT
	tyWhiteCeilingNorth:			Type_LED;
	tyWhiteCeilingSouth:			Type_LED;
	tyWhiteWorkplateNorth:		Type_LED;
	tyWhiteWorkplateSouth:		Type_LED;
	tyWhiteTableNorth:			Type_LED;
	tyWhiteTableSouth:			Type_LED;
END_VAR
(*LED light white ceiling north*)
PRG_LED_SINGLECOLOR(
	i_bSwitchOn:= FALSE,
	i_bSwitchOff:= FALSE,
	i_bSwitchOnOff:= FALSE,
	i_iSceneValue:= ,
	io_TypeLED:= tyWhiteCeilingNorth);

(*LED light white ceiling south*)
PRG_LED_SINGLECOLOR(
	i_bSwitchOn:= FALSE,
	i_bSwitchOff:= FALSE,
	i_bSwitchOnOff:= FALSE,
	i_iSceneValue:= ,
	io_TypeLED:= tyWhiteCeilingSouth);

(*LED light white workplate north*)
PRG_LED_SINGLECOLOR(
	i_bSwitchOn:= FALSE,
	i_bSwitchOff:= FALSE,
	i_bSwitchOnOff:= FALSE,
	i_iSceneValue:= ,
	io_TypeLED:= tyWhiteWorkplateNorth);

(*LED light white workplate south*)
PRG_LED_SINGLECOLOR(
	i_bSwitchOn:= FALSE,
	i_bSwitchOff:= FALSE,
	i_bSwitchOnOff:= FALSE,
	i_iSceneValue:= ,
	io_TypeLED:= tyWhiteWorkplateSouth);

(*LED light white table north*)
PRG_LED_SINGLECOLOR(
	i_bSwitchOn:= FALSE,
	i_bSwitchOff:= FALSE,
	i_bSwitchOnOff:= FALSE,
	i_iSceneValue:= ,
	io_TypeLED:= tyWhiteTableNorth);

(*LED light white table south*)
PRG_LED_SINGLECOLOR(
	i_bSwitchOn:= FALSE,
	i_bSwitchOff:= FALSE,
	i_bSwitchOnOff:= FALSE,
	i_iSceneValue:= ,
	io_TypeLED:= tyWhiteTableSouth);

(*relay for power supply*)
DO_NN_K05 :=	tyWhiteCeilingNorth.bLight OR tyWhiteCeilingSouth.bLight OR tyWhiteWorkplateNorth.bLight OR
				tyWhiteWorkplateSouth.bLight OR tyWhiteTableNorth.bLight OR tyWhiteTableSouth.bLight;

(*DMX communication*)
arrDMXProcessData[40] := tyWhiteCeilingNorth.Brightness;
arrDMXProcessData[41] := tyWhiteCeilingSouth.Brightness;
arrDMXProcessData[42] := tyWhiteWorkplateNorth.Brightness;
arrDMXProcessData[43] := tyWhiteWorkplateSouth.Brightness;
arrDMXProcessData[44] := tyWhiteTableNorth.Brightness;
arrDMXProcessData[45] := tyWhiteTableSouth.Brightness;
END_PROGRAM

(* POU FC_04_ZIMMER, ST *)
PROGRAM FC_04_ZIMMER
VAR PERSISTENT
	tyWhiteCeiling:			Type_LED;
	tyWhiteReserve1:			Type_LED;
	tyWhiteReserve2:			Type_LED;
	tyWhiteReserve3:			Type_LED;
	tyWhiteSZCeiling:			Type_LED;
	tyWhiteSZBed:			Type_LED;
	tyWhiteSZReadLeft:		Type_LED;
	tyWhiteSZReadRight:		Type_LED;
END_VAR
(*LED light white ceiling*)
PRG_LED_SINGLECOLOR(
	i_bSwitchOn:= FALSE,
	i_bSwitchOff:= FALSE,
	i_bSwitchOnOff:= FALSE,
	i_iSceneValue:= ,
	io_TypeLED:= tyWhiteCeiling);

(*LED light white spare*)
PRG_LED_SINGLECOLOR(
	i_bSwitchOn:= FALSE,
	i_bSwitchOff:= FALSE,
	i_bSwitchOnOff:= FALSE,
	i_iSceneValue:= ,
	io_TypeLED:= tyWhiteReserve1);

(*LED light white spare*)
PRG_LED_SINGLECOLOR(
	i_bSwitchOn:= FALSE,
	i_bSwitchOff:= FALSE,
	i_bSwitchOnOff:= FALSE,
	i_iSceneValue:= ,
	io_TypeLED:= tyWhiteReserve2);

(*LED light white spare*)
PRG_LED_SINGLECOLOR(
	i_bSwitchOn:= FALSE,
	i_bSwitchOff:= FALSE,
	i_bSwitchOnOff:= FALSE,
	i_iSceneValue:= ,
	io_TypeLED:= tyWhiteReserve3);

(*LED light white SZ ceiling*)
PRG_LED_SINGLECOLOR(
	i_bSwitchOn:= FALSE,
	i_bSwitchOff:= FALSE,
	i_bSwitchOnOff:= FALSE,
	i_iSceneValue:= ,
	io_TypeLED:= tyWhiteSZCeiling);

(*LED light white SZ bed*)
PRG_LED_SINGLECOLOR(
	i_bSwitchOn:= FALSE,
	i_bSwitchOff:= FALSE,
	i_bSwitchOnOff:= FALSE,
	i_iSceneValue:= ,
	io_TypeLED:= tyWhiteSZBed);

(*LED light white SZ read left*)
PRG_LED_SINGLECOLOR(
	i_bSwitchOn:= FALSE,
	i_bSwitchOff:= FALSE,
	i_bSwitchOnOff:= FALSE,
	i_iSceneValue:= ,
	io_TypeLED:= tyWhiteSZReadLeft);

(*LED light white SZ read right*)
PRG_LED_SINGLECOLOR(
	i_bSwitchOn:= FALSE,
	i_bSwitchOff:= FALSE,
	i_bSwitchOnOff:= FALSE,
	i_iSceneValue:= ,
	io_TypeLED:= tyWhiteSZReadRight);

(*relay for power supply*)
DO_NN_K06 :=	tyWhiteCeiling.bLight OR tyWhiteReserve1.bLight OR tyWhiteReserve2.bLight OR
				tyWhiteReserve3.bLight OR tyWhiteSZCeiling.bLight OR tyWhiteSZBed.bLight OR
				tyWhiteSZReadLeft.bLight OR tyWhiteSZReadRight.bLight;

(*DMX communication*)
arrDMXProcessData[60] := tyWhiteCeiling.Brightness;
arrDMXProcessData[61] := tyWhiteReserve1.Brightness;
arrDMXProcessData[62] := tyWhiteReserve2.Brightness;
arrDMXProcessData[63] := tyWhiteReserve3.Brightness;
arrDMXProcessData[64] := tyWhiteSZCeiling.Brightness;
arrDMXProcessData[65] := tyWhiteSZBed.Brightness;
arrDMXProcessData[66] := tyWhiteSZReadLeft.Brightness;
arrDMXProcessData[67] := tyWhiteSZReadRight.Brightness;
END_PROGRAM

(* POU FC_05_WC_GANG, ST *)
PROGRAM FC_05_WC_GANG
VAR PERSISTENT
	tyWhiteWC:			Type_LED;
	tyWhiteGarderobe:		Type_LED;
	tyWhiteAreaKitchen:	Type_LED;
	tyWhiteReserve1:		Type_LED;
	tyWhiteMirror:			Type_LED;
	tyWhiteReserve2:		Type_LED;
	tyWhiteReserve3:		Type_LED;
	tyWhiteReserve4:		Type_LED;

END_VAR
VAR
	fbLightBathroom: FB_Light;
END_VAR
(*LED light white WC*)
PRG_LED_SINGLECOLOR(
	i_bSwitchOn:= FALSE,
	i_bSwitchOff:= FALSE,
	i_bSwitchOnOff:= DI_S08,
	i_iSceneValue:= ,
	io_TypeLED:= tyWhiteWC);

(*LED light white Garderobe*)
PRG_LED_SINGLECOLOR(
	i_bSwitchOn:= FALSE,
	i_bSwitchOff:= FALSE,
	i_bSwitchOnOff:= FALSE,
	i_iSceneValue:= ,
	io_TypeLED:= tyWhiteGarderobe);

(*LED light white Bereich Küche*)
PRG_LED_SINGLECOLOR(
	i_bSwitchOn:= FALSE,
	i_bSwitchOff:= FALSE,
	i_bSwitchOnOff:= FALSE,
	i_iSceneValue:= ,
	io_TypeLED:= tyWhiteAreaKitchen);

(*LED light white spare*)
PRG_LED_SINGLECOLOR(
	i_bSwitchOn:= FALSE,
	i_bSwitchOff:= FALSE,
	i_bSwitchOnOff:= FALSE,
	i_iSceneValue:= ,
	io_TypeLED:= tyWhiteReserve1);

(*LED light white Spiegel*)
PRG_LED_SINGLECOLOR(
	i_bSwitchOn:= FALSE,
	i_bSwitchOff:= FALSE,
	i_bSwitchOnOff:= FALSE,
	i_iSceneValue:= ,
	io_TypeLED:= tyWhiteMirror);

(*LED light white Reserve*)
PRG_LED_SINGLECOLOR(
	i_bSwitchOn:= FALSE,
	i_bSwitchOff:= FALSE,
	i_bSwitchOnOff:= FALSE,
	i_iSceneValue:= ,
	io_TypeLED:= tyWhiteReserve2);

(*LED light white Reserve*)
PRG_LED_SINGLECOLOR(
	i_bSwitchOn:= FALSE,
	i_bSwitchOff:= FALSE,
	i_bSwitchOnOff:= FALSE,
	i_iSceneValue:= ,
	io_TypeLED:= tyWhiteReserve3);

(*LED light white Reserve*)
PRG_LED_SINGLECOLOR(
	i_bSwitchOn:= FALSE,
	i_bSwitchOff:= FALSE,
	i_bSwitchOnOff:= FALSE,
	i_iSceneValue:= ,
	io_TypeLED:= tyWhiteReserve4);

(*relay for power supply*)
DO_NN_K07 :=	tyWhiteWC.bLight OR tyWhiteGarderobe.bLight OR tyWhiteAreaKitchen.bLight OR
				tyWhiteReserve1.bLight OR tyWhiteMirror.bLight OR tyWhiteReserve2.bLight OR
				tyWhiteReserve3.bLight OR tyWhiteReserve4.bLight;

(*light bathroom*)
fbLightBathroom(bOn:=FALSE , bOff:=FALSE , bToggle:=DI_S11 , bLight=> DO_NN_K08);

(*DMX communication*)
arrDMXProcessData[80] := tyWhiteWC.Brightness;
arrDMXProcessData[81] := tyWhiteGarderobe.Brightness;
arrDMXProcessData[82] := tyWhiteAreaKitchen.Brightness;
arrDMXProcessData[83] := tyWhiteReserve1.Brightness;
arrDMXProcessData[84] := tyWhiteMirror.Brightness;
arrDMXProcessData[85] := tyWhiteReserve2.Brightness;
arrDMXProcessData[86] := tyWhiteReserve3.Brightness;
arrDMXProcessData[87] := tyWhiteReserve4.Brightness;
END_PROGRAM

(* POU Weather/YAHOO_WEATHER_test, CFC *)
PROGRAM YAHOO_WEATHER_test
VAR
	IP_C: IP_C;
	S_BUF: NETWORK_BUFFER;
	R_BUF: NETWORK_BUFFER;
	IP_CONTROL_1: IP_CONTROL;
	activate: BOOL;
	done: BOOL;
	busy: BOOL;
	error_c: DWORD;
	error_t: BYTE;
	YAHOO_WEATHER: YAHOO_WEATHER;
	YW_DATA: YAHOO_WEATHER_DATA;
	CLK_PRG: CLK_PRG;
	YAHOO_WEATHER_DESC_GE: YAHOO_WEATHER_DESC_GE;
	YAHOO_WEATHER_ICON_OSCAT: YAHOO_WEATHER_ICON_OSCAT;
END_VAR
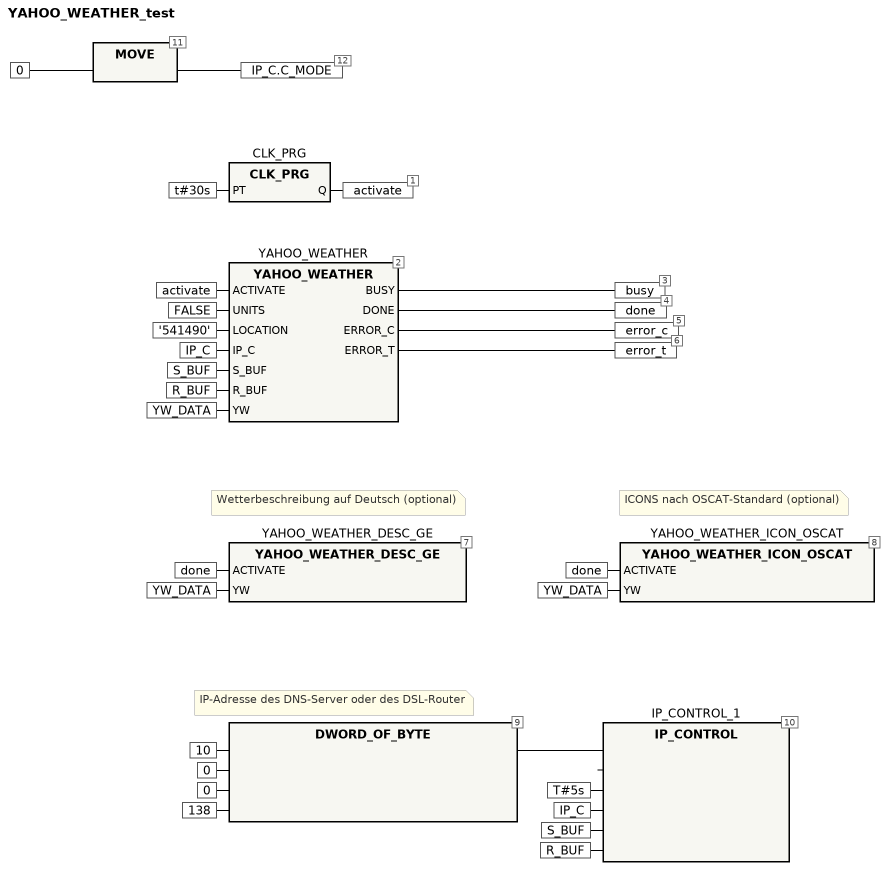
_CFC_ (* Continuous Function Chart, elements in execution order *)
#0 CLK_PRG:CLK_PRG(PT: t#30s)
#1 activate <= #0.Q
#2 YAHOO_WEATHER:YAHOO_WEATHER(ACTIVATE: activate, UNITS: FALSE, LOCATION: '541490', IP_C: IP_C, S_BUF: S_BUF, R_BUF: R_BUF, YW: YW_DATA)
#3 busy <= #2.BUSY
#4 done <= #2.DONE
#5 error_c <= #2.ERROR_C
#6 error_t <= #2.ERROR_T
#7 YAHOO_WEATHER_DESC_GE:YAHOO_WEATHER_DESC_GE(ACTIVATE: done, YW: YW_DATA)
#8 YAHOO_WEATHER_ICON_OSCAT:YAHOO_WEATHER_ICON_OSCAT(ACTIVATE: done, YW: YW_DATA)
#9 DWORD_OF_BYTE(10, 0, 0, 138)
#10 IP_CONTROL_1:IP_CONTROL(#9, -, T#5s, IP_C, S_BUF, R_BUF)
(* ICONS nach OSCAT-Standard (optional) *)
(* IP-Adresse des DNS-Server oder des DSL-Router *)
(* Wetterbeschreibung auf Deutsch (optional) *)
#11 MOVE(0)
#12 IP_C.C_MODE <= #11
_END_CFC_
END_PROGRAM

(* POU Weather/WORLD_WEATHER_test, CFC *)
PROGRAM WORLD_WEATHER_test
VAR
	IP_C: IP_C;
	S_BUF: NETWORK_BUFFER;
	R_BUF: NETWORK_BUFFER;
	IP_CONTROL_1: IP_CONTROL;
	activate: BOOL := TRUE;
	done: BOOL;
	busy: BOOL;
	error_c: DWORD;
	error_t: BYTE;
	latitude: REAL := 48.21;
	longitude: REAL := 16.37;
	WORLD_WEATHER: WORLD_WEATHER;
	WW_DATA: WORLD_WEATHER_DATA;
	CLK_PRG: CLK_PRG;
	WORLD_WEATHER_DESC_GE: WORLD_WEATHER_DESC_GE;
	WORLD_WEATHER_ICON_OSCAT: WORLD_WEATHER_ICON_OSCAT;
END_VAR
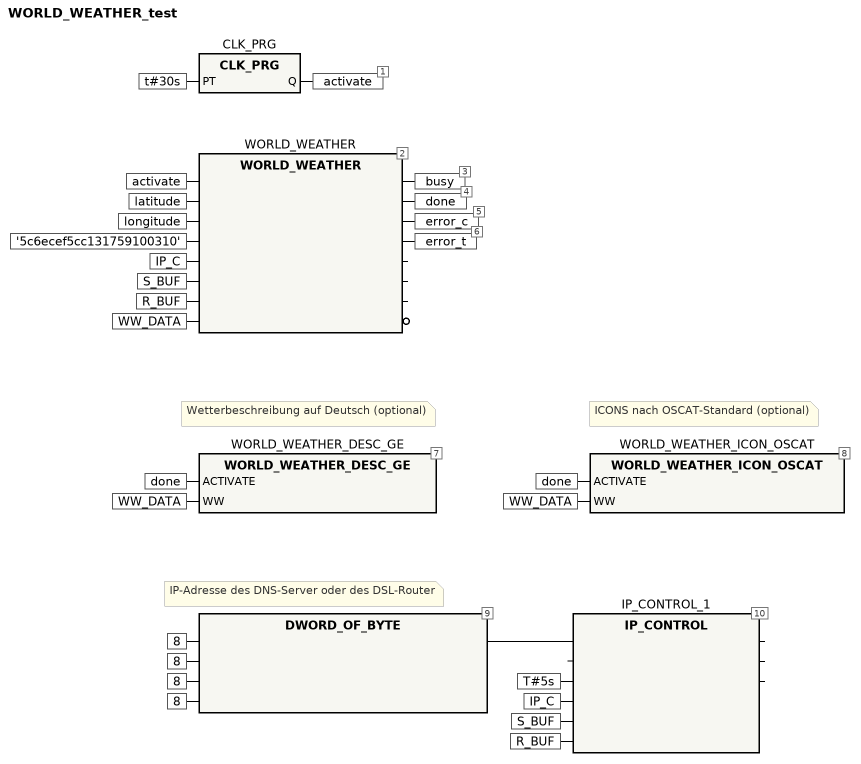
_CFC_ (* Continuous Function Chart, elements in execution order *)
#0 CLK_PRG:CLK_PRG(PT: t#30s)
#1 activate <= #0.Q
#2 WORLD_WEATHER:WORLD_WEATHER(activate, latitude, longitude, '5c6ecef5cc131759100310', IP_C, S_BUF, R_BUF, WW_DATA)
#3 busy <= #2.out 1
#4 done <= #2.out 2
#5 error_c <= #2.out 3
#6 error_t <= #2.out 4
#7 WORLD_WEATHER_DESC_GE:WORLD_WEATHER_DESC_GE(ACTIVATE: done, WW: WW_DATA)
#8 WORLD_WEATHER_ICON_OSCAT:WORLD_WEATHER_ICON_OSCAT(ACTIVATE: done, WW: WW_DATA)
#9 DWORD_OF_BYTE(8, 8, 8, 8)
#10 IP_CONTROL_1:IP_CONTROL(#9, -, T#5s, IP_C, S_BUF, R_BUF)
(* ICONS nach OSCAT-Standard (optional) *)
(* IP-Adresse des DNS-Server oder des DSL-Router *)
(* Wetterbeschreibung auf Deutsch (optional) *)
_END_CFC_
END_PROGRAM
